{attribute 'qualified_only'}
{attribute 'strict'}
TYPE CETA_Result_e :
(
	OK := 1,
	NOK := 2
)USINT;
END_TYPE

(* stored: Version 1.1.0.1, ProductVersion 3.1.4024.6
   DUT CETA_Result_e: Id {4d576c91-b9f3-4e86-a06d-73520521f7ac} *)
